// TwinCAT 3 PLC project PPMCheckout
// ProgramVersion: 3.1.4022.7
// libraries:
//   LCLS General, * (SLAC)
//   lcls-twincat-motion, * (SLAC)
//   lcls2-cc-lib, * (SLAC)
//   Tc2_Standard, * (Beckhoff Automation GmbH)
//   Tc2_System, * (Beckhoff Automation GmbH)
//   Tc3_Module, * (Beckhoff Automation GmbH)
//   VisuDialogs, * (System)
// project tree:
//   DUTs/ DUT_MotionStage_Extras.TcDUT (not stored)
//   / GlobalTextList.TcGTLO, PlcTask.TcTTO (not stored), Visualization Manager.TcVMO (not stored)
//   POUs/ Main.TcPOU
//   VISUs/ TextListPPMStates.TcTLO (not stored), Visualization.TcVIS (not stored), VISU_MotionStage.TcVIS
// real-time tasks:
//   TASK PlcTask: cycle T#10ms, priority 20, ADS port 350
// motion (NC):
// I/O:
//   DEVICE Device 1 (EtherCAT)
// variable links:
//   PPMCheckout Instance <-> Device 1 (EtherCAT)/Term 3 (EK1100)/TST-EL2004
//     PlcTask Outputs/Main.M1.bBrakeRelease <-> Channel 1/Output
//     PlcTask Outputs/Main.fbPPM.fbGige.bGigePower <-> Channel 2/Output
//   PPMCheckout Instance <-> Device 1 (EtherCAT)/Term 3 (EK1100)/TST-EL3062
//     PlcTask Inputs/Main.fbPPM.fbPowerMeter.iVoltageINT <-> AI Standard Channel 1/Value
//   PPMCheckout Instance <-> Device 1 (EtherCAT)/Term 3 (EK1100)/TST-EL3314
//     PlcTask Inputs/Main.fbPPM.fbPowerMeter.fbThermoCouple.bError <-> TC Inputs Channel 1/Status/Error
//     PlcTask Inputs/Main.fbPPM.fbPowerMeter.fbThermoCouple.bOverrange <-> TC Inputs Channel 1/Status/Overrange
//     PlcTask Inputs/Main.fbPPM.fbPowerMeter.fbThermoCouple.bUnderrange <-> TC Inputs Channel 1/Status/Underrange
//     PlcTask Inputs/Main.fbPPM.fbPowerMeter.fbThermoCouple.iRaw <-> TC Inputs Channel 1/Value
//     PlcTask Inputs/Main.fbPPM.fbYagThermoCouple.bError <-> TC Inputs Channel 2/Status/Error
//     PlcTask Inputs/Main.fbPPM.fbYagThermoCouple.bOverrange <-> TC Inputs Channel 2/Status/Overrange
//     PlcTask Inputs/Main.fbPPM.fbYagThermoCouple.bUnderrange <-> TC Inputs Channel 2/Status/Underrange
//     PlcTask Inputs/Main.fbPPM.fbYagThermoCouple.iRaw <-> TC Inputs Channel 2/Value
//   PPMCheckout Instance <-> Device 1 (EtherCAT)/Term 3 (EK1100)/TST-EL4004
//     PlcTask Outputs/Main.fbPPM.fbGige.iIlluminatorINT <-> AO Outputs Channel 1/Analog output
//   PPMCheckout Instance <-> Device 1 (EtherCAT)/Term 3 (EK1100)/TST-EL5042
//     PlcTask Inputs/Main.iRawEncoder <-> FB Inputs Channel 1/Position
//   PPMCheckout Instance <-> Device 1 (EtherCAT)/Term 3 (EK1100)/TST-EL7041
//     PlcTask Inputs/Main.M1.bLimitBackwardEnable <-> STM Status/Status/Digital input 2
//     PlcTask Inputs/Main.M1.bLimitForwardEnable <-> STM Status/Status/Digital input 1
//   PPMCheckout Instance <-> NC-Task 1 SAF/Axes/Axis 1
//     PlcTask Inputs/Main.M1.Axis.NcToPlc <-> Outputs/ToPlc
//     PlcTask Outputs/Main.M1.Axis.PlcToNc <-> Inputs/FromPlc

// ---- POUs/Main.TcPOU
PROGRAM Main
VAR
	{attribute 'pytmc' := 'pv: TST:PPM:MMS'}
	{attribute 'TcLinkTo' := '.bLimitForwardEnable  := TIIB[TST-EL7041]^STM Status^Status^Digital input 1;
	                          .bLimitBackwardEnable := TIIB[TST-EL7041]^STM Status^Status^Digital input 2;
	                          .bBrakeRelease        := TIIB[TST-EL2004]^Channel 1^Output'}
	M1: DUT_MotionStage;
	
	{attribute 'pytmc' := '
		pv: TST:PPM
		io: io
	'}
	{attribute 'TcLinkTo' := '.fbGige.iIlluminatorINT := TIIB[TST-EL4004]^AO Outputs Channel 1^Analog output;
	                          .fbGige.bGigePower := TIIB[TST-EL2004]^Channel 2^Output;
							  .fbPowerMeter.iVoltageINT := TIIB[TST-EL3062]^AI Standard Channel 1^Value;
							  .fbPowerMeter.fbThermoCouple.bError := TIIB[TST-EL3314]^TC Inputs Channel 1^Status^Error;
							  .fbPowerMeter.fbThermoCouple.bUnderrange := TIIB[TST-EL3314]^TC Inputs Channel 1^Status^Underrange;
							  .fbPowerMeter.fbThermoCouple.bOverrange := TIIB[TST-EL3314]^TC Inputs Channel 1^Status^Overrange;
							  .fbPowerMeter.fbThermoCouple.iRaw := TIIB[TST-EL3314]^TC Inputs Channel 1^Value;
							  .fbYagThermoCouple.bError := TIIB[TST-EL3314]^TC Inputs Channel 2^Status^Error;
							  .fbYagThermoCouple.bUnderrange := TIIB[TST-EL3314]^TC Inputs Channel 2^Status^Underrange;
							  .fbYagThermoCouple.bOverrange := TIIB[TST-EL3314]^TC Inputs Channel 2^Status^Overrange;
							  .fbYagThermoCouple.iRaw := TIIB[TST-EL3314]^TC Inputs Channel 2^Value'}
	fbPPM: FB_PPM;
	
	M1_Extras: DUT_MotionStage_Extras;
	
	iRawEncoder AT %I*: ULINT;
	iAdjustedEncoder: ULINT;
END_VAR

fbPPM(
	stYStage := M1,
	fPolished := -50,
	fFrosted := -40,
	fPower := -30,
	fOut := -20);

M1_Extras.bVisuHighLim := NOT M1.bAllForwardEnable;
M1_Extras.bVisuLowLim := NOT M1.bAllBackwardEnable;
	
iAdjustedEncoder := LINT_TO_ULINT(-ULINT_TO_LINT(iRawEncoder));

END_PROGRAM

// ---- GlobalTextList.TcGTLO
TEXTLIST GlobalTextList
  167 = '%f'
  888 = '%X'
  532 = '+'
  526 = '-'
  884 = '0 = Default Acceleration'
  886 = '0 = Default Deceleration'
  883 = 'Acceleration: %f'
  667 = 'Cam Power'
  530 = 'Clear'
  524 = 'Control'
  665 = 'Controls'
  168 = 'Current Position'
  885 = 'Deceleration: %f'
  889 = 'Error Code'
  887 = 'Error:'
  528 = 'GO'
  529 = 'GO to set position'
  169 = 'High Limit Hit Indicator'
  666 = 'Illuminator: %f %'
  166 = 'Low Limit Hit Indicator'
  826 = 'Motor'
  170 = 'Moving:'
  663 = 'PM Temp: %f C'
  830 = 'Power Meter: %f V'
  827 = 'PPM'
  828 = 'Raw count: %d'
  829 = 'Readbacks'
  525 = 'Set Position'
  533 = 'Settings'
  924 = 'State: '
  960 = 'State:  %s'
  905 = 'State: %i'
  165 = 'Status'
  527 = 'Step Size'
  531 = 'STOP'
  534 = 'Velocity: %f'
  664 = 'Yag Temp: %f C'
END_TEXTLIST

// ---- VISUs/VISU_MotionStage.TcVIS
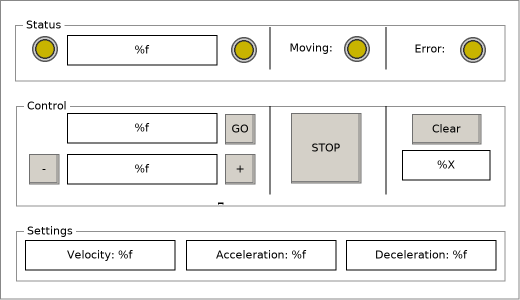
VISUALIZATION VISU_MotionStage  // 520x300
VAR_IN_OUT
	VisuMotionStage: DUT_MotionStage;
	Extras: DUT_MotionStage_Extras;
END_VAR
    GroupBox (15,17 490x64), "Status"
        Lamp1 (15,17 30x30), tooltip "Low Limit Hit Indicator", variable: Extras.bVisuLowLim, style: Lamp-Lamp1-Yellow
        Rectangle (52,18 150x30), "%f", tooltip "Current Position", text variable: VisuMotionStage.stAxisStatus.fActPosition
        Lamp1 (214,18 30x30), tooltip "High Limit Hit Indicator", variable: Extras.bVisuHighLim, style: Lamp-Lamp1-Yellow
        Lamp1 (327,17 30x30), variable: VisuMotionStage.bBusy, style: Lamp-Lamp1-Yellow
        Label (262,16 68x30), "Moving:"
        Line (371,52) (371,10)
        Lamp1 (443,18 30x30), variable: VisuMotionStage.bError, style: Lamp-Lamp1-Yellow
    Rectangle (218,203 5x0)
    GroupBox (16,98 489x108), "Control"
        Rectangle (51,15 150x30), "%f", tooltip "Set Position", text variable: VisuMotionStage.fPosition
            OnMouseDown: write the text variable via Default
        Button (13,56 30x30), "-"
            OnMouseDown: execute {
                VisuMotionStage.nCommand := 3;
                VisuMotionStage.fPosition := VisuMotionStage.stAxisStatus.fActPosition - Extras.fVisuStep;
                VisuMotionStage.bExecute := TRUE;
            }
        Rectangle (51,56 150x30), "%f", tooltip "Step Size", text variable: Extras.fVisuStep
            OnMouseDown: write the text variable via Default
        Button (209,16 30x30), "GO", tooltip "GO to set position"
            OnMouseDown: execute { VisuMotionStage.nCommand := 3; VisuMotionStage.bExecute := TRUE; }
        Line (254,96) (254,8)
        Line (370,96) (370,8)
        Button (396,16 69x30), "Clear"
            tap VisuMotionStage.bReset
        Button (275,15 70x70), "STOP", tooltip "GO to set position"
            OnMouseDown: execute { VisuMotionStage.bExecute := FALSE; }
        Button (209,56 30x30), "+"
            OnMouseDown: execute {
                VisuMotionStage.nCommand := 3;
                VisuMotionStage.fPosition := VisuMotionStage.stAxisStatus.fActPosition + Extras.fVisuStep;
                VisuMotionStage.bExecute := TRUE;
            }
    GroupBox (16,223 489x58), "Settings"
        Rectangle (9,17 150x30), "Velocity: %f", text variable: VisuMotionStage.fVelocity
            OnMouseDown: write the text variable via Default
        Rectangle (170,17 150x30), "Acceleration: %f", tooltip "0 = Default Acceleration", text variable: VisuMotionStage.fAcceleration
            OnMouseDown: write the text variable via Default
        Rectangle (330,17 150x30), "Deceleration: %f", tooltip "0 = Default Deceleration", text variable: VisuMotionStage.fDeceleration
            OnMouseDown: write the text variable via Default
    Line (270,69) (270,27)
    Label (396,34 68x30), "Error:"
    Rectangle (402,150 88x30), "%X", tooltip "Error Code", text variable: VisuMotionStage.nErrorId
END_VISUALIZATION
